VISUALIZATION LeftRobotStats  // 2x2
END_VISUALIZATION

(* stored: Version 1.1.0.1, ProductVersion 3.1.4024.15
   Visu LeftRobotStats: Id {f767bf11-0e75-4eda-9995-f3229458b862} *)
